// TwinCAT 3 PLC project ProjectMain
// ProgramVersion: 3.1.4023.0
// libraries:
//   Tc2_ControllerToolbox, * (Beckhoff Automation GmbH)
//   Tc2_Math, * (Beckhoff Automation GmbH)
//   Tc2_MC2, * (Beckhoff Automation GmbH)
//   Tc2_MC2_Drive, * (Beckhoff Automation GmbH)
//   Tc2_NCI, * (Beckhoff Automation GmbH)
//   Tc2_NcKinematicTransformation, * (Beckhoff Automation GmbH)
//   Tc2_PlcInterpolation, * (Beckhoff Automation GmbH)
//   Tc2_Standard, * (Beckhoff Automation GmbH)
//   Tc2_System, * (Beckhoff Automation GmbH)
//   Tc2_Utilities, * (Beckhoff Automation GmbH)
//   Tc3_McCollisionAvoidance, * (Beckhoff Automation GmbH)
//   Tc3_McCoordinatedMotion, * (Beckhoff Automation GmbH)
//   Tc3_Module, * (Beckhoff Automation GmbH)
//   Tc3_Vision, * (Beckhoff Automation GmbH)
//   Tc3_XTS_Utility, * (Beckhoff Automation GmbH)
// project tree:
//   DUTs/ DeltaCommands_typ.TcDUT, DeltaMotionParameters_typ.TcDUT, DeltaState_enum.TcDUT, ElevatorState_enum.TcDUT, MachineOperationMode.TcDUT, MainCommands_typ.TcDUT, MainStateAxis_enum.TcDUT, MainState_enum.TcDUT, MotionParameters_typ.TcDUT, MoverCommandType_enum.TcDUT, MoverState_enum.TcDUT, MoveState_t.TcDUT, PickPars_typ.TcDUT, Pucks.TcDUT, SystemCommands_typ.TcDUT, Vector3Position_typ.TcDUT, Visu_typ.TcDUT, Coords.TcDUT, XYParams_typ.TcDUT
//   GVLs/ GVL.TcGVL, GVL_Conveyer.TcGVL, GVL_Vision.TcGVL, GVL_XTS.TcGVL, GVL_XY.TcGVL
//   ITFs/ iDelta.TcIO, iRoute.TcIO
//   / Main1_1.TcTTO, Main2_1.TcTTO, Main3_1.TcTTO, Main4_1.TcTTO, Main5_1.TcTTO
//   Station1%28Codian%29/ Faults1.TcPOU (not stored), fbLoadMoves.TcPOU (not stored), Forces1.TcPOU (not stored), Main1.TcPOU (not stored), Reset1.TcPOU (not stored), Sequence1.TcPOU (not stored)
//   Station1%28Codian%29/Functions/ Delta.TcPOU (not stored), FB_PuckPicked.TcPOU (not stored), Route.TcPOU (not stored)
//   Station2%28XYmover%29/ Faults2.TcPOU (not stored), Forces2.TcPOU (not stored), Main2.TcPOU (not stored), Reset2.TcPOU (not stored), Sequence2.TcPOU (not stored)
//   Station2%28XYmover%29/XY_FBs/ FB_AddAllAxes.TcPOU (not stored), FB_ConveyerTimer.TcPOU (not stored), FB_PowerAll.TcPOU (not stored), FB_ResetAllAxis.TcPOU (not stored), FB_StopAll.TcPOU (not stored)
//   Station3%28Conveyor%29/ Faults3.TcPOU (not stored), Forces3.TcPOU (not stored), Main3.TcPOU (not stored), Reset3.TcPOU (not stored), Sequence3.TcPOU (not stored)
//   Station3%28Conveyor%29/Functions/ FB_ClearConveyer.TcPOU (not stored), FB_ConveyerStop.TcPOU (not stored), FB_PowerConveyer.TcPOU (not stored)
//   Station4%28xts1%29/ Faults4.TcPOU (not stored), Forces4.TcPOU (not stored), Main4.TcPOU (not stored), Reset4.TcPOU (not stored), Sequence4.TcPOU (not stored)
//   Station5%28xts2%29/ Faults5.TcPOU (not stored), Forces5.TcPOU (not stored), Main5.TcPOU (not stored), Reset5.TcPOU (not stored), Sequence5.TcPOU (not stored)
//   Station6%28Vision%29/ Faults6.TcPOU (not stored), Forces6.TcPOU (not stored), Main6.TcPOU (not stored), Reset6.TcPOU (not stored), Sequence6.TcPOU (not stored)
// real-time tasks:
//   TASK PlcTask: cycle T#10ms, priority 20, ADS port 350
//   TASK VnTask ADS (Camera1): cycle T#10ms, priority 16, ADS port 354
//   TASK VnTask ImgAcq (Camera1): cycle T#1ms, priority 10, ADS port 353
//   TASK Job Task: cycle default, priority 32
//   TASK Main1: cycle T#1ms, priority 2, ADS port 351
//   TASK Main2: cycle T#10ms, priority 3, ADS port 355
//   TASK Main3: cycle T#10ms, priority 5, ADS port 356
//   TASK Main4: cycle T#10ms, priority 6, ADS port 357
//   TASK Main5: cycle T#10ms, priority 7, ADS port 358
// motion (NC):
//   TASK NC-Task 1 SAF: cycle T#500us, priority 4, ADS port 501
//   TASK NC-Task 1 SVB: cycle T#10ms, priority 8, ADS port 511
//   AXIS Delta ACS A (id 10)
//     General: UnitName=°
//     Dynamic: Acceleration=2367.9, Deceleration=2367.9, Jerk=7103.7
//     Velo: RefSearch=15.78603, RefSync=15.78603, SlowManual=78.93015, FastManual=473.5809, Fast=1578.603, Maximum=1578.6
//     OtherSettings: AllowMotionCmdToSlave=true
//     encoder EncType=19
//       EncPara: ScaleFactorNumerator=360, ScaleFactorDenominator=23068672, Offset=-24.7313, Inverse=true, MaxCount=#xffffffff
//     drive DrvType=16
//       DrvPara: Inverse=true, MaxCount=#xffffffff, DriveControlDWord=#x00020100
//         Analog: VeloReferenz=1736.4633, TorqueSetpointScale=10, ScaleFactorActTorque=0.1
//         TimeComp: TaskDelayCycles=1
//     controller CtrType=1
//       CtrPara: PriorControlFactor=1
//         Observer: BandWidth=20
//   AXIS Delta ACS B (id 11)
//     General: UnitName=°
//     Dynamic: Acceleration=2367.9, Deceleration=2367.9, Jerk=7103.71
//     Velo: RefSearch=15.78603, RefSync=15.78603, SlowManual=78.93015, FastManual=473.5809, Fast=1578.603, Maximum=1578.6
//     OtherSettings: AllowMotionCmdToSlave=true
//     encoder EncType=19
//       EncPara: ScaleFactorNumerator=360, ScaleFactorDenominator=23068672, Offset=1838.2737, Inverse=true, MaxCount=#xffffffff
//     drive DrvType=16
//       DrvPara: Inverse=true, MaxCount=#xffffffff, DriveControlDWord=#x00020100
//         Analog: VeloReferenz=1736.4633, TorqueSetpointScale=10, ScaleFactorActTorque=0.1
//         TimeComp: TaskDelayCycles=1
//     controller CtrType=1
//       CtrPara: PriorControlFactor=1
//         Observer: BandWidth=20
//   AXIS Delta ACS C (id 12)
//     General: UnitName=°
//     Dynamic: Acceleration=2367.9045, Deceleration=2367.9045, Jerk=7103.7135
//     Velo: RefSearch=15.78603, RefSync=15.78603, SlowManual=78.93015, FastManual=473.5809, Fast=1578.603, Maximum=1578.603
//     OtherSettings: AllowMotionCmdToSlave=true
//     encoder EncType=19
//       EncPara: ScaleFactorNumerator=360, ScaleFactorDenominator=23068672, Offset=9.7019, Inverse=true, MaxCount=#xffffffff
//     drive DrvType=16
//       DrvPara: Inverse=true, MaxCount=#xffffffff, DriveControlDWord=#x00020100
//         Analog: VeloReferenz=1736.4633, TorqueSetpointScale=10, ScaleFactorActTorque=0.1
//         TimeComp: TaskDelayCycles=1
//     controller CtrType=1
//       CtrPara: PriorControlFactor=1
//         Observer: BandWidth=20
//   AXIS Delta MCS X (id 5)
//     Dynamic: Acceleration=12900, Deceleration=12900, Jerk=286914
//     OtherSettings: AllowMotionCmdToSlave=true
//     encoder EncType=1
//       SoftEndMinControl: Enable=true, Range=-100
//       SoftEndMaxControl: Enable=true, Range=100
//     drive DrvType=5
//       Analog: VeloReferenz=500, TorqueSetpointScale=10, ScaleFactorActTorque=0.1
//       TimeComp: TaskDelayCycles=1
//     controller CtrType=1
//       CtrPara: PriorControlFactor=1
//         Observer: BandWidth=20
//   AXIS Delta MCS Y (id 6)
//     Dynamic: Acceleration=13125, Deceleration=13125, Jerk=275625
//     OtherSettings: AllowMotionCmdToSlave=true
//     encoder EncType=1
//       SoftEndMinControl: Enable=true, Range=-80
//       SoftEndMaxControl: Enable=true, Range=150
//     drive DrvType=5
//       Analog: VeloReferenz=500, TorqueSetpointScale=10, ScaleFactorActTorque=0.1
//       TimeComp: TaskDelayCycles=1
//     controller CtrType=1
//       CtrPara: PriorControlFactor=1
//         Observer: BandWidth=20
//   AXIS Delta MCS Z (id 7)
//     Dynamic: Acceleration=15100, Deceleration=15100, Jerk=223539
//     OtherSettings: AllowMotionCmdToSlave=true
//     encoder EncType=1
//       EncPara: Offset=-250
//         SoftEndMinControl: Range=-60
//         SoftEndMaxControl: Enable=true, Range=25
//     drive DrvType=5
//       Analog: VeloReferenz=500, TorqueSetpointScale=10, ScaleFactorActTorque=0.1
//       TimeComp: TaskDelayCycles=1
//     controller CtrType=1
//       CtrPara: PriorControlFactor=1
//         Observer: BandWidth=20
//   AXIS Y (id 1)
//     Dynamic: Acceleration=540.1395, Deceleration=540.1395, Jerk=1620.4185
//     Velo: RefSearch=3.60093, RefSync=3.60093, SlowManual=18.00465, FastManual=108.0279, Fast=360.093, Maximum=360.093
//     OtherSettings: AllowMotionCmdToSlave=true
//     encoder EncType=19
//       EncPara: ScaleFactorNumerator=4, ScaleFactorDenominator=1048576, Offset=7764.81834411621, MaxCount=#xffffffff, ReferenceSystem=1
//         SoftEndMinControl: Enable=true
//         SoftEndMaxControl: Enable=true, Range=385
//     drive DrvType=16
//       DrvPara: MaxCount=#xffffffff, DriveControlDWord=#x00020100
//         Analog: VeloReferenz=396.1023, VeloScale=32, TorqueSetpointScale=10, ScaleFactorActTorque=0.1
//         TimeComp: TaskDelayCycles=1
//     controller CtrType=1
//       CtrPara: PriorControlFactor=1
//         Observer: BandWidth=20
//   AXIS X (id 2)
//     Dynamic: Acceleration=540.9, Deceleration=540.9, Jerk=1622.7
//     Velo: RefSearch=3.606, RefSync=3.606, SlowManual=18.03, FastManual=108.18, Fast=360.6, Maximum=360.6
//     OtherSettings: AllowMotionCmdToSlave=true
//     encoder EncType=19
//       EncPara: ScaleFactorNumerator=4, ScaleFactorDenominator=1048576, MaxCount=#xffffffff, ReferenceSystem=3
//         SoftEndMinControl: Enable=true
//         SoftEndMaxControl: Enable=true, Range=200
//     drive DrvType=16
//       DrvPara: MaxCount=#xffffffff, DriveControlDWord=#x00020100
//         Analog: VeloReferenz=396.66, VeloScale=32, TorqueSetpointScale=10, ScaleFactorActTorque=0.1
//         TimeComp: TaskDelayCycles=1
//     controller CtrType=1
//       CtrPara: PriorControlFactor=1
//         Observer: BandWidth=20
//   AXIS X Slave (id 3)
//     Dynamic: Acceleration=524.2, Deceleration=524.2, Jerk=1572.6
//     Velo: RefSearch=3.49466666666667, RefSync=3.49466666666667, SlowManual=17.4733333333333, FastManual=104.84, Fast=349.466666666667, Maximum=349.466666666667
//     OtherSettings: AllowMotionCmdToSlave=true
//     encoder EncType=19
//       EncPara: ScaleFactorNumerator=4, ScaleFactorDenominator=1048576, Offset=-2512.61434173584, MaxCount=#xffffffff, ReferenceSystem=3
//         SoftEndMinControl: Enable=true
//         SoftEndMaxControl: Enable=true, Range=200
//     drive DrvType=16
//       DrvPara: MaxCount=#xffffffff, DriveControlDWord=#x00020100
//         Analog: VeloReferenz=384.413333333333, VeloScale=32, TorqueSetpointScale=10, ScaleFactorActTorque=0.1
//         TimeComp: TaskDelayCycles=1
//     controller CtrType=1
//       CtrPara: PriorControlFactor=1
//         Observer: BandWidth=20
//   AXIS ConveyorAxis (id 4)
//     General: UnitName=°
//     Dynamic: AccelerationMaximum=48963.411, DecelerationMaximum=48963.411, Acceleration=48681, Deceleration=48681, Jerk=146043
//     Velo: RefSearch=324.54, RefSync=324.54, SlowManual=1622.7, FastManual=9736.2, Fast=32454, Maximum=32454
//     OtherSettings: AllowMotionCmdToSlave=true
//     encoder EncType=19
//       EncPara: ScaleFactorNumerator=360, ScaleFactorDenominator=1048576, MaxCount=#xffffffff
//     drive DrvType=16
//       DrvPara: MaxCount=#xffffffff, DriveControlDWord=#x00020100
//         Analog: VeloReferenz=35699.4, VeloScale=32, TorqueSetpointScale=10, ScaleFactorActTorque=0.1
//         TimeComp: TaskDelayCycles=1
//     controller CtrType=1
//       CtrPara: PriorControlFactor=1
//         PosDiffControl: Enable=false, Range=25
//         Observer: BandWidth=20
// I/O:
//   DEVICE Device 3 (EtherCAT), AmsNetId 169.254.124.141.4.1
//     Term 1 (EK1100) [EK1100 EtherCAT Coupler (2A E-Bus)]
//       Term 2 (EL1918) [EL1918, 8Ch. Safety Input 24V, TwinSAFE]
//         modules: Module 2 (FSLOGIC)
//       Term 3 (EL1008) [EL1008 8Ch. Dig. Input 24V, 3ms]
//       Term 4 (EL2904) [EL2904, 4 Ch. Safety Output 24V, 0.5A, TwinSAFE]
//         modules: Module 1 (FSOES), Module 2 (DO)
//       Term 5 (EL2008) [EL2008 8Ch. Dig. Output 24V, 0.5A]
//       Term 6 (EL7201-9014) [EL7201-9014 1Ch. MDP742 Servo motor output stage with OCT (50V, 4A)  and STO input]
//         startup 32785:27 := 23150000 // DRV Motor Settings / Motor speed limitation
//         startup 32784:19 := B200 // DRV Amplifier Settings / Current loop proportional gain
//         startup 32784:18 := 0500 // DRV Amplifier Settings / Current loop integral time
//         startup 32784:21 := 25000000 // DRV Amplifier Settings / Velocity loop proportional gain
//         startup 32784:20 := 96000000 // DRV Amplifier Settings / Velocity loop integral time
//         startup 32768:1 := 00 // FB Settings / Invert feedback direction
//       Term 7 (EL7211-9014) [EL7211-9014 1Ch. MDP742 Servo motor output stage with OCT (50V, 4.5A RMS) and STO input]
//         startup 32785:21 := 0E01 // DRV Motor Settings / Commutation offset
//         startup 32786:19 := F401 // DRV Brake Settings / Emergency application timeout
//         startup 32784:51 := 0A00 // DRV Amplifier Settings / Stand still window
//         startup 32785:27 := 21150000 // DRV Motor Settings / Motor speed limitation
//         startup 32784:19 := B200 // DRV Amplifier Settings / Current loop proportional gain
//         startup 32784:18 := 0500 // DRV Amplifier Settings / Current loop integral time
//         startup 32784:21 := 48000000 // DRV Amplifier Settings / Velocity loop proportional gain
//         startup 32784:20 := 96000000 // DRV Amplifier Settings / Velocity loop integral time
//         startup 32768:1 := 00 // FB Settings / Invert feedback direction
//       Term 22 (EL7211-9014) [EL7211-9014 1Ch. MDP742 Servo motor output stage with OCT (50V, 4.5A RMS) and STO input]
//         startup 32784:18 := 0A00
//         startup 32784:19 := 6400
//         startup 32784:20 := 32000000
//         startup 32784:21 := 96000000
//         startup 32784:51 := 0A00
//         startup 32785:17 := 98210000
//         startup 32785:18 := 960A0000
//         startup 32785:19 := 03
//         startup 32785:21 := 0E01
//         startup 32785:22 := 46000000
//         startup 32785:24 := 39000000
//         startup 32785:25 := 0F00
//         startup 32785:27 := FF120000
//         startup 32785:45 := 5501
//         startup 32786:17 := 0800
//         startup 32786:18 := 0E00
//         startup 32786:19 := F401
//       Term 9 (EL7211-9014) [EL7211-9014 1Ch. MDP742 Servo motor output stage with OCT (50V, 4.5A RMS) and STO input]
//         startup 32785:21 := 0E01 // DRV Motor Settings / Commutation offset
//         startup 32786:19 := F401 // DRV Brake Settings / Emergency application timeout
//         startup 32784:51 := 0A00 // DRV Amplifier Settings / Stand still window
//         startup 32785:27 := 21150000 // DRV Motor Settings / Motor speed limitation
//         startup 32784:19 := B200 // DRV Amplifier Settings / Current loop proportional gain
//         startup 32784:18 := 0500 // DRV Amplifier Settings / Current loop integral time
//         startup 32784:21 := 48000000 // DRV Amplifier Settings / Velocity loop proportional gain
//         startup 32784:20 := 96000000 // DRV Amplifier Settings / Velocity loop integral time
//         startup 32768:1 := 00 // FB Settings / Invert feedback direction
//       Term 13 (EL9011) [EL9011 End Terminal]
//     Term 10 (AX8620-0000-0103) [AX8620-0000-0103]
//       Drive 11 (AX8108-0100-0104) [AX8108-0100-0104 (1Ch. 8A servo axis, STO)]
//         modules: Device, Device, Device, Device, Device, Device, Device, Device, Device, Device, Device (Safety), Device, Device, Device, Device, Device, Device, Device, Device, Device, Device, Device, Device, Device, Device, Device, Device, Device, Device, Device, Device, Ch A, Ch A, Ch A, Ch A, Ch A, Ch A, Ch A, Ch A, Ch A, Ch A, Ch A, Ch A, Ch A, Ch A, Ch A, Ch A, Ch A, Ch A, Ch A, Ch A, Ch A, Ch A, Ch A, Ch A, Ch A, Ch A, Ch A
//         startup 12992:1 := 414D383033312D78467830 // Ch A Motor parameters / Configured motor type
//         startup 24768:0 := FEFF // Ch A Interpolation sub mode select
//         startup 13000:5 := 0200 // Ch A Motor thermal model / Reaction
//         startup 13000:6 := 0000C841 // Ch A Motor thermal model / Partial fraction factor
//         startup 12992:12 := 00A00C46 // Ch A Motor parameters / Motor rated speed
//         startup 12992:13 := 2731A83F // Ch A Motor parameters / Motor rated torque
//         startup 24694:0 := 7A050000 // Ch A Motor standstill torque
//         startup 24800:0 := D007 // Ch A Positive torque/force limit value
//         startup 24801:0 := D007 // Ch A Negative torque/force limit value
//         startup 12288:6 := 4158383130382D303130302D30303030 // Ch A AxisMain parameters / Configured drive type
//         startup 12867:1 := CDCC4C40 // Ch A TorqueCtrl parameters / Configured channel rated current
//         startup 12867:2 := 9A991941 // Ch A TorqueCtrl parameters / Configured channel peak current
//         startup 24672:0 := 08 // Ch A Modes of operation
//         startup 12864:1 := 60CE3E42 // Ch A TorqueCtrl parameters mappable / Torque control proportional gain q
//         startup 12864:2 := 8A0E7C39 // Ch A TorqueCtrl parameters mappable / Torque control integral action time q
//         startup 12608:1 := 9C67B13C // Ch A VeloCtrl parameters mappable / Velocity control proportional gain
//         startup 12608:2 := 6F12033C // Ch A VeloCtrl parameters mappable / Velocity control integral action time
//         startup 12608:3 := 00980546 // Ch A VeloCtrl parameters mappable / Bipolar velocity limit value
//         startup 12992:15 := 0100 // Ch A Motor parameters / Motor temperature sensor connection
//         startup 12611:4 := 0400 // Ch A VeloCtrl observer / Observer type
//         startup 24672:0 := 08 // Ch A Modes of operation
//         startup 12296:2 := 00 // Ch A AxisMain parameters encoder polarity / Primary encoder actual values
//       Drive 12 (AX8206-0210-0104) [AX8206-0210-0104 (2Ch. 6A servo axis, safe-motion, multi-FB)]
//         modules: Device, Device, Device, Device, Device, Device, Device, Device, Device, Device, Device (Safety), Device, Device, Device, Device, Device, Device, Device, Device, Device, Device, Device, Device, Device, Device, Device, Device, Device, Device, Device, Device, Ch A, Ch A, Ch A, Ch A, Ch A, Ch A, Ch A, Ch A, Ch A, Ch A, Ch A, Ch A, Ch A, Ch A, Ch A, Ch A, Ch A, Ch A, Ch A, Ch A, Ch A, Ch A, Ch A, Ch A, Ch A, Ch A, Ch B, Ch B, Ch B, Ch B, Ch B, Ch B, Ch B, Ch B, Ch B, Ch B, Ch B, Ch B, Ch B, Ch B, Ch B, Ch B, Ch B, Ch B, Ch B, Ch B, Ch B, Ch B, Ch B, Ch B, Ch B, Ch B
//         startup 12992:1 := 414D383033312D78467830 // Ch A Motor parameters / Configured motor type
//         startup 24768:0 := FEFF // Ch A Interpolation sub mode select
//         startup 13000:5 := 0200 // Ch A Motor thermal model / Reaction
//         startup 13000:6 := 0000C841 // Ch A Motor thermal model / Partial fraction factor
//         startup 12992:12 := 00A00C46 // Ch A Motor parameters / Motor rated speed
//         startup 12992:13 := 2731A83F // Ch A Motor parameters / Motor rated torque
//         startup 24694:0 := 7A050000 // Ch A Motor standstill torque
//         startup 24800:0 := D007 // Ch A Positive torque/force limit value
//         startup 24801:0 := D007 // Ch A Negative torque/force limit value
//         startup 12288:6 := 4158383230362D303231302D30303030 // Ch A AxisMain parameters / Configured drive type
//         startup 12867:1 := CDCC4C40 // Ch A TorqueCtrl parameters / Configured channel rated current
//         startup 12867:2 := 9A991941 // Ch A TorqueCtrl parameters / Configured channel peak current
//         startup 24672:0 := 08 // Ch A Modes of operation
//         startup 12864:1 := 60CE3E42 // Ch A TorqueCtrl parameters mappable / Torque control proportional gain q
//         startup 12864:2 := 8A0E7C39 // Ch A TorqueCtrl parameters mappable / Torque control integral action time q
//         startup 12608:1 := 9C67B13C // Ch A VeloCtrl parameters mappable / Velocity control proportional gain
//         startup 12608:2 := 6F12033C // Ch A VeloCtrl parameters mappable / Velocity control integral action time
//         startup 12608:3 := 00980546 // Ch A VeloCtrl parameters mappable / Bipolar velocity limit value
//         startup 12992:15 := 0100 // Ch A Motor parameters / Motor temperature sensor connection
//         startup 12611:4 := 0400 // Ch A VeloCtrl observer / Observer type
//         startup 24672:0 := 08 // Ch A Modes of operation
//         startup 12296:2 := 00 // Ch A AxisMain parameters encoder polarity / Primary encoder actual values
//         startup 14016:1 := 414D383033312D78467830 // Ch B Motor parameters / Configured motor type
//         startup 26816:0 := FEFF // Ch B Interpolation sub mode select
//         startup 14024:5 := 0200 // Ch B Motor thermal model / Reaction
//         startup 14024:6 := 0000C841 // Ch B Motor thermal model / Partial fraction factor
//         startup 14016:12 := 00A00C46 // Ch B Motor parameters / Motor rated speed
//         startup 14016:13 := 2731A83F // Ch B Motor parameters / Motor rated torque
//         startup 26742:0 := 7A050000 // Ch B Motor standstill torque
//         startup 26848:0 := D007 // Ch B Positive torque/force limit value
//         startup 26849:0 := D007 // Ch B Negative torque/force limit value
//         startup 13312:6 := 4158383230362D303231302D30303030 // Ch B AxisMain parameters / Configured drive type
//         startup 13891:1 := CDCC4C40 // Ch B TorqueCtrl parameters / Configured channel rated current
//         startup 13891:2 := 9A991941 // Ch B TorqueCtrl parameters / Configured channel peak current
//         startup 26720:0 := 08 // Ch B Modes of operation
//         startup 13888:1 := 60CE3E42 // Ch B TorqueCtrl parameters mappable / Torque control proportional gain q
//         startup 13888:2 := 8A0E7C39 // Ch B TorqueCtrl parameters mappable / Torque control integral action time q
//         startup 13632:1 := 9C67B13C // Ch B VeloCtrl parameters mappable / Velocity control proportional gain
//         startup 13632:2 := 6F12033C // Ch B VeloCtrl parameters mappable / Velocity control integral action time
//         startup 13632:3 := 00980546 // Ch B VeloCtrl parameters mappable / Bipolar velocity limit value
//         startup 14016:15 := 0100 // Ch B Motor parameters / Motor temperature sensor connection
//         startup 13635:4 := 0400 // Ch B VeloCtrl observer / Observer type
//         startup 26720:0 := 08 // Ch B Modes of operation
//         startup 13320:2 := 00 // Ch B AxisMain parameters encoder polarity / Primary encoder actual values
//       Term 14 (EL9011) [EL9011 End Terminal]
//   DEVICE Device 1 (EtherCAT Automation Protocol), AmsNetId 169.254.124.141.2.1
//     Box 8 (Publisher)
//     Box 15 (Subscriber)
// variable links:
//   Device 3 (EtherCAT) <-> Device 3 (EtherCAT)/Term 1 (EK1100)/Term 2 (EL1918)
//     Term 1 (EK1100)/Term 4 (EL2904)/Module 1 (FSOES)/RxPDO/FSOE <-> ConnectionInputs/Message_4 TxPDO
//     Term 10 (AX8620-0000-0103)/Drive 12 (AX8206-0210-0104)/Device (Safety)/FSoE Slave Connection 1 Slave Message/FSOE <-> ConnectionOutputs/Message_6 RxPDO
//   Device 3 (EtherCAT) <-> Device 3 (EtherCAT)/Term 1 (EK1100)/Term 4 (EL2904)
//     Term 1 (EK1100)/Term 2 (EL1918)/ConnectionOutputs/Message_4 RxPDO <-> Module 1 (FSOES)/TxPDO/FSOE
//   Device 3 (EtherCAT) <-> Device 3 (EtherCAT)/Term 10 (AX8620-0000-0103)
//     Term 10 (AX8620-0000-0103)/Drive 11 (AX8108-0100-0104)/Device/DeviceMain Outputs/Power supply controlword <-> PSM Controlword for axis/Controlword for axis
//     Term 10 (AX8620-0000-0103)/Drive 12 (AX8206-0210-0104)/Device/DeviceMain Outputs/Power supply controlword <-> PSM Controlword for axis/Controlword for axis
//   Device 3 (EtherCAT) <-> Device 3 (EtherCAT)/Term 10 (AX8620-0000-0103)/Drive 11 (AX8108-0100-0104)
//     Term 1 (EK1100)/Term 2 (EL1918)/ConnectionInputs/Message_5 TxPDO <-> Device (Safety)/FSoE Slave Connection 1 Master Message/FSOE
//     Term 1 (EK1100)/Term 2 (EL1918)/ConnectionOutputs/Message_5 RxPDO <-> Device (Safety)/FSoE Slave Connection 1 Slave Message/FSOE
//   Device 3 (EtherCAT) <-> Device 3 (EtherCAT)/Term 10 (AX8620-0000-0103)/Drive 12 (AX8206-0210-0104)
//     Term 1 (EK1100)/Term 2 (EL1918)/ConnectionInputs/Message_6 TxPDO <-> Device (Safety)/FSoE Slave Connection 1 Master Message/FSOE
//   NC-Task 1 SAF/Axes/ConveyorAxis <-> Device 3 (EtherCAT)/Term 1 (EK1100)/Term 9 (EL7211-9014)
//     Drive/Inputs/In/nDataIn1 <-> DRV Following error actual value/Following error actual value
//     Drive/Inputs/In/nDcOutputTime <-> InfoData/DcOutputShift
//     Drive/Inputs/In/nState1 <-> DRV Statusword/Statusword
//     Drive/Inputs/In/nState2 <-> DRV Statusword/Statusword @bit 8
//     Drive/Inputs/In/nState4 @bit 1 <-> WcState/InputToggle
//     Drive/Inputs/In/nState4 <-> WcState/WcState
//     Drive/Outputs/Out/nCtrl1 <-> DRV Controlword/Controlword
//     Drive/Outputs/Out/nCtrl2 <-> DRV Controlword/Controlword @bit 8
//     Drive/Outputs/Out/nDataOut1 <-> DRV Target position/Target position
//     Drive/Outputs/Out/nDataOut2 <-> DRV Target velocity/Target velocity
//     Enc/Inputs/In/nDataIn1 <-> FB Position/Position
//     Enc/Inputs/In/nDcInputTime <-> InfoData/DcInputShift
//     Enc/Inputs/In/nState4 @bit 1 <-> WcState/InputToggle
//     Enc/Inputs/In/nState4 <-> WcState/WcState
//   NC-Task 1 SAF/Axes/Delta ACS A <-> Device 3 (EtherCAT)/Term 10 (AX8620-0000-0103)/Drive 11 (AX8108-0100-0104)
//     Drive/Inputs/In/nDataIn1 <-> Ch A/Ch A PositionControl Inputs/Ch A Following error actual value
//     Drive/Inputs/In/nDcOutputTime <-> InfoData/DcOutputShift
//     Drive/Inputs/In/nState1 <-> Ch A/Ch A AxisMain Inputs/Ch A Statusword
//     Drive/Inputs/In/nState2 <-> Ch A/Ch A AxisMain Inputs/Ch A Statusword @bit 8
//     Drive/Inputs/In/nState4 @bit 1 <-> WcState/InputToggle0
//     Drive/Inputs/In/nState4 <-> WcState/WcState0
//     Drive/Outputs/Out/nCtrl1 <-> Ch A/Ch A AxisMain Outputs/Ch A Controlword
//     Drive/Outputs/Out/nCtrl2 <-> Ch A/Ch A AxisMain Outputs/Ch A Controlword @bit 8
//     Drive/Outputs/Out/nDataOut1 <-> Ch A/Ch A Interpolator Outputs/Ch A Target position
//     Drive/Outputs/Out/nDataOut2 <-> Ch A/Ch A Interpolator Outputs/Ch A Target velocity
//     Enc/Inputs/In/nDataIn1 <-> Ch A/Ch A AxisMain Inputs/Ch A Position actual value
//     Enc/Inputs/In/nDcInputTime <-> InfoData/DcInputShift
//     Enc/Inputs/In/nState2 @bit 5 <-> Ch A/Ch A AxisMain Inputs/Position actual value invalid
//     Enc/Inputs/In/nState4 @bit 1 <-> WcState/InputToggle0
//     Enc/Inputs/In/nState4 <-> WcState/WcState0
//   NC-Task 1 SAF/Axes/Delta ACS B <-> Device 3 (EtherCAT)/Term 10 (AX8620-0000-0103)/Drive 12 (AX8206-0210-0104)
//     Drive/Inputs/In/nDataIn1 <-> Ch A/Ch A PositionControl Inputs/Ch A Following error actual value
//     Drive/Inputs/In/nDcOutputTime <-> InfoData/DcOutputShift
//     Drive/Inputs/In/nState1 <-> Ch A/Ch A AxisMain Inputs/Ch A Statusword
//     Drive/Inputs/In/nState2 <-> Ch A/Ch A AxisMain Inputs/Ch A Statusword @bit 8
//     Drive/Inputs/In/nState4 @bit 1 <-> WcState/InputToggle0
//     Drive/Inputs/In/nState4 <-> WcState/WcState0
//     Drive/Outputs/Out/nCtrl1 <-> Ch A/Ch A AxisMain Outputs/Ch A Controlword
//     Drive/Outputs/Out/nCtrl2 <-> Ch A/Ch A AxisMain Outputs/Ch A Controlword @bit 8
//     Drive/Outputs/Out/nDataOut1 <-> Ch A/Ch A Interpolator Outputs/Ch A Target position
//     Drive/Outputs/Out/nDataOut2 <-> Ch A/Ch A Interpolator Outputs/Ch A Target velocity
//     Enc/Inputs/In/nDataIn1 <-> Ch A/Ch A AxisMain Inputs/Ch A Position actual value
//     Enc/Inputs/In/nDcInputTime <-> InfoData/DcInputShift
//     Enc/Inputs/In/nState2 @bit 5 <-> Ch A/Ch A AxisMain Inputs/Position actual value invalid
//     Enc/Inputs/In/nState4 @bit 1 <-> WcState/InputToggle0
//     Enc/Inputs/In/nState4 <-> WcState/WcState0
//   NC-Task 1 SAF/Axes/Delta ACS C <-> Device 3 (EtherCAT)/Term 10 (AX8620-0000-0103)/Drive 12 (AX8206-0210-0104)
//     Drive/Inputs/In/nDataIn1 <-> Ch B/Ch B PositionControl Inputs/Ch B Following error actual value
//     Drive/Inputs/In/nDcOutputTime <-> InfoData/DcOutputShift
//     Drive/Inputs/In/nState1 <-> Ch B/Ch B AxisMain Inputs/Ch B Statusword
//     Drive/Inputs/In/nState2 <-> Ch B/Ch B AxisMain Inputs/Ch B Statusword @bit 8
//     Drive/Inputs/In/nState4 @bit 1 <-> WcState/InputToggle0
//     Drive/Inputs/In/nState4 <-> WcState/WcState0
//     Drive/Outputs/Out/nCtrl1 <-> Ch B/Ch B AxisMain Outputs/Ch B Controlword
//     Drive/Outputs/Out/nCtrl2 <-> Ch B/Ch B AxisMain Outputs/Ch B Controlword @bit 8
//     Drive/Outputs/Out/nDataOut1 <-> Ch B/Ch B Interpolator Outputs/Ch B Target position
//     Drive/Outputs/Out/nDataOut2 <-> Ch B/Ch B Interpolator Outputs/Ch B Target velocity
//     Enc/Inputs/In/nDataIn1 <-> Ch B/Ch B AxisMain Inputs/Ch B Position actual value
//     Enc/Inputs/In/nDcInputTime <-> InfoData/DcInputShift
//     Enc/Inputs/In/nState2 @bit 5 <-> Ch B/Ch B AxisMain Inputs/Position actual value invalid
//     Enc/Inputs/In/nState4 @bit 1 <-> WcState/InputToggle0
//     Enc/Inputs/In/nState4 <-> WcState/WcState0
//   NC-Task 1 SAF/Axes/X <-> Device 3 (EtherCAT)/Term 1 (EK1100)/Term 7 (EL7211-9014)
//     Drive/Inputs/In/nDataIn1 <-> DRV Following error actual value/Following error actual value
//     Drive/Inputs/In/nDcOutputTime <-> InfoData/DcOutputShift
//     Drive/Inputs/In/nState1 <-> DRV Statusword/Statusword
//     Drive/Inputs/In/nState2 <-> DRV Statusword/Statusword @bit 8
//     Drive/Inputs/In/nState4 @bit 1 <-> WcState/InputToggle
//     Drive/Inputs/In/nState4 <-> WcState/WcState
//     Drive/Outputs/Out/nCtrl1 <-> DRV Controlword/Controlword
//     Drive/Outputs/Out/nCtrl2 <-> DRV Controlword/Controlword @bit 8
//     Drive/Outputs/Out/nDataOut1 <-> DRV Target position/Target position
//     Drive/Outputs/Out/nDataOut2 <-> DRV Target velocity/Target velocity
//     Enc/Inputs/In/nDataIn1 <-> FB Position/Position
//     Enc/Inputs/In/nDcInputTime <-> InfoData/DcInputShift
//     Enc/Inputs/In/nState4 @bit 1 <-> WcState/InputToggle
//     Enc/Inputs/In/nState4 <-> WcState/WcState
//   NC-Task 1 SAF/Axes/X Slave <-> Device 3 (EtherCAT)/Term 1 (EK1100)/Term 22 (EL7211-9014)
//     Drive/Inputs/In/nDataIn1 <-> DRV Following error actual value/Following error actual value
//     Drive/Inputs/In/nDcOutputTime <-> InfoData/DcOutputShift
//     Drive/Inputs/In/nState1 <-> DRV Statusword/Statusword
//     Drive/Inputs/In/nState2 <-> DRV Statusword/Statusword @bit 8
//     Drive/Inputs/In/nState4 @bit 1 <-> WcState/InputToggle
//     Drive/Inputs/In/nState4 <-> WcState/WcState
//     Drive/Outputs/Out/nCtrl1 <-> DRV Controlword/Controlword
//     Drive/Outputs/Out/nCtrl2 <-> DRV Controlword/Controlword @bit 8
//     Drive/Outputs/Out/nDataOut1 <-> DRV Target position/Target position
//     Drive/Outputs/Out/nDataOut2 <-> DRV Target velocity/Target velocity
//     Enc/Inputs/In/nDataIn1 <-> FB Position/Position
//     Enc/Inputs/In/nDcInputTime <-> InfoData/DcInputShift
//     Enc/Inputs/In/nState4 @bit 1 <-> WcState/InputToggle
//     Enc/Inputs/In/nState4 <-> WcState/WcState
//   NC-Task 1 SAF/Axes/Y <-> Device 3 (EtherCAT)/Term 1 (EK1100)/Term 6 (EL7201-9014)
//     Drive/Inputs/In/nDataIn1 <-> DRV Following error actual value/Following error actual value
//     Drive/Inputs/In/nDcOutputTime <-> InfoData/DcOutputShift
//     Drive/Inputs/In/nState1 <-> DRV Statusword/Statusword
//     Drive/Inputs/In/nState2 <-> DRV Statusword/Statusword @bit 8
//     Drive/Inputs/In/nState4 @bit 1 <-> WcState/InputToggle
//     Drive/Inputs/In/nState4 <-> WcState/WcState
//     Drive/Outputs/Out/nCtrl1 <-> DRV Controlword/Controlword
//     Drive/Outputs/Out/nCtrl2 <-> DRV Controlword/Controlword @bit 8
//     Drive/Outputs/Out/nDataOut1 <-> DRV Target position/Target position
//     Drive/Outputs/Out/nDataOut2 <-> DRV Target velocity/Target velocity
//     Enc/Inputs/In/nDataIn1 <-> FB Position/Position
//     Enc/Inputs/In/nDcInputTime <-> InfoData/DcInputShift
//     Enc/Inputs/In/nState4 @bit 1 <-> WcState/InputToggle
//     Enc/Inputs/In/nState4 <-> WcState/WcState
//   ProjectMain/ProjectMain Instance <-> Device 1 (EtherCAT Automation Protocol)/Box 15 (Subscriber)
//     Main1_1 Inputs/GVL_XTS.mover0InPosition <-> mover0InPosition/Inputs/VarData
//     Main2_1 Inputs/GVL_XTS.moversInPosition[1] <-> moversInPosition/Inputs/VarData[1]
//     Main2_1 Inputs/GVL_XTS.moversInPosition[2] <-> moversInPosition/Inputs/VarData[2]
//     Main2_1 Inputs/GVL_XTS.moversInPosition[3] <-> moversInPosition/Inputs/VarData[3]
//     Main5_1 Inputs/GVL_XTS.moversReleased[1] <-> moversReleased/Inputs/VarData[1]
//     Main5_1 Inputs/GVL_XTS.moversReleased[2] <-> moversReleased/Inputs/VarData[2]
//     Main5_1 Inputs/GVL_XTS.moversReleased[3] <-> moversReleased/Inputs/VarData[3]
//   ProjectMain/ProjectMain Instance <-> Device 1 (EtherCAT Automation Protocol)/Box 8 (Publisher)
//     Main1_1 Outputs/GVL_XTS.bDeltaRelease <-> bDeltaRelease/Outputs/VarData
//     Main2_1 Outputs/GVL_XTS.moversRelease <-> moversRelease/Outputs/VarData[1]
//     Main2_1 Outputs/GVL_XTS.moversRelease @bit 8 <-> moversRelease/Outputs/VarData[2]
//     Main2_1 Outputs/GVL_XTS.moversRelease @bit 16 <-> moversRelease/Outputs/VarData[3]
//     Main4_1 Outputs/GVL_XTS.XTS_Disable <-> XTS_Disable/Outputs/VarData
//     Main4_1 Outputs/GVL_XTS.XTS_Enable <-> XTS_Enable/Outputs/VarData
//     Main4_1 Outputs/GVL_XTS.XTS_Start <-> XTS_Start/Outputs/VarData
//     Main4_1 Outputs/GVL_XTS.XTS_Stop <-> XTS_Stop/Outputs/VarData
//   ProjectMain/ProjectMain Instance <-> Device 3 (EtherCAT)/Term 1 (EK1100)/Term 3 (EL1008)
//     Main1_1 Inputs/GVL_Conveyer.bSensor <-> Channel 7/GVL_Conveyer.bSensor
//   ProjectMain/ProjectMain Instance <-> Device 3 (EtherCAT)/Term 1 (EK1100)/Term 5 (EL2008)
//     Main1_1 Outputs/Main1.Sequence1.Delta.AirVariable <-> Channel 8/Main1.Sequence.Delta.AirVariable
//     Main2_1 Outputs/GVL_XY.bAirEnable <-> Channel 2/GantryVacuum
//     Main2_1 Outputs/GVL_XY.bPullUp <-> Channel 4/GrantryPushUp
//     Main2_1 Outputs/GVL_XY.bPushDown <-> Channel 6/GantryPushDown
//   ProjectMain/ProjectMain Instance <-> NC-Task 1 SAF/Axes/ConveyorAxis
//     Main2_1 Inputs/GVL_Conveyer.ConveyerAxis.NcToPlc <-> Outputs/ToPlc
//     Main2_1 Outputs/GVL_Conveyer.ConveyerAxis.PlcToNc <-> Inputs/FromPlc
//   ProjectMain/ProjectMain Instance <-> NC-Task 1 SAF/Axes/Delta ACS A
//     Main1_1 Inputs/Main1.Sequence1.Delta.ACS_A_REF.NcToPlc <-> Outputs/ToPlc
//     Main1_1 Outputs/Main1.Sequence1.Delta.ACS_A_REF.PlcToNc <-> Inputs/FromPlc
//   ProjectMain/ProjectMain Instance <-> NC-Task 1 SAF/Axes/Delta ACS B
//     Main1_1 Inputs/Main1.Sequence1.Delta.ACS_B_REF.NcToPlc <-> Outputs/ToPlc
//     Main1_1 Outputs/Main1.Sequence1.Delta.ACS_B_REF.PlcToNc <-> Inputs/FromPlc
//   ProjectMain/ProjectMain Instance <-> NC-Task 1 SAF/Axes/Delta ACS C
//     Main1_1 Inputs/Main1.Sequence1.Delta.ACS_C_REF.NcToPlc <-> Outputs/ToPlc
//     Main1_1 Outputs/Main1.Sequence1.Delta.ACS_C_REF.PlcToNc <-> Inputs/FromPlc
//   ProjectMain/ProjectMain Instance <-> NC-Task 1 SAF/Axes/Delta MCS X
//     Main1_1 Inputs/Main1.Sequence1.Delta.MCS_X_REF.NcToPlc <-> Outputs/ToPlc
//     Main1_1 Outputs/Main1.Sequence1.Delta.MCS_X_REF.PlcToNc <-> Inputs/FromPlc
//   ProjectMain/ProjectMain Instance <-> NC-Task 1 SAF/Axes/Delta MCS Y
//     Main1_1 Inputs/Main1.Sequence1.Delta.MCS_Y_REF.NcToPlc <-> Outputs/ToPlc
//     Main1_1 Outputs/Main1.Sequence1.Delta.MCS_Y_REF.PlcToNc <-> Inputs/FromPlc
//   ProjectMain/ProjectMain Instance <-> NC-Task 1 SAF/Axes/Delta MCS Z
//     Main1_1 Inputs/Main1.Sequence1.Delta.MCS_Z_REF.NcToPlc <-> Outputs/ToPlc
//     Main1_1 Outputs/Main1.Sequence1.Delta.MCS_Z_REF.PlcToNc <-> Inputs/FromPlc
//   ProjectMain/ProjectMain Instance <-> NC-Task 1 SAF/Axes/X
//     Main2_1 Inputs/GVL_XY.stAxis[1].NcToPlc <-> Outputs/ToPlc
//     Main2_1 Outputs/GVL_XY.stAxis[1].PlcToNc <-> Inputs/FromPlc
//   ProjectMain/ProjectMain Instance <-> NC-Task 1 SAF/Axes/X Slave
//     Main2_1 Inputs/GVL_XY.stSlaveAxis[1].NcToPlc <-> Outputs/ToPlc
//     Main2_1 Outputs/GVL_XY.stSlaveAxis[1].PlcToNc <-> Inputs/FromPlc
//   ProjectMain/ProjectMain Instance <-> NC-Task 1 SAF/Axes/Y
//     Main2_1 Inputs/GVL_XY.stAxis[2].NcToPlc <-> Outputs/ToPlc
//     Main2_1 Outputs/GVL_XY.stAxis[2].PlcToNc <-> Inputs/FromPlc
//   ProjectMain/ProjectMain Instance <-> NC-Task 1 SAF/Channel_Kinnematics
//     Main1_1 Inputs/Main1.Sequence1.Delta.internalKinChanNCtoPLC <-> Outputs/Main1.Sequence.Delta.internalKinChanNCtoPLC
//     Main1_1 Outputs/Main1.Sequence1.Delta.internalKinChanPLCtoNC <-> Inputs/Main1.Sequence.Delta.internalKinChanPLCtoNC
//   ProjectMain/ProjectMain Instance <-> NC-Task 1 SAF/Objects/Delta MC CM
//     Main1_1 Inputs/Main1.Sequence1.Delta.internalCMGroup.NcToPlc <-> Group Outputs/ToPLC
//     Main1_1 Outputs/Main1.Sequence1.Delta.internalCMGroup.PlcToNc <-> Group Inputs/FromPLC
//   ProjectMain/ProjectMain Instance <-> NC-Task 1 SAF/Objects/Gantry MC CM
//     Main5_1 Inputs/GVL_XY.stGroupRef.NcToPlc <-> Group Outputs/ToPLC
//     Main5_1 Outputs/GVL_XY.stGroupRef.PlcToNc <-> Group Inputs/FromPLC

CONFIGURATION ProjectMain
    RESOURCE PLC ON TwinCAT3
        TASK Main1_1(INTERVAL := T#1ms, PRIORITY := 2);
        TASK Main2_1(INTERVAL := T#10ms, PRIORITY := 3);
        TASK Main3_1(INTERVAL := T#10ms, PRIORITY := 5);
        TASK Main4_1(INTERVAL := T#10ms, PRIORITY := 6);
        TASK Main5_1(INTERVAL := T#10ms, PRIORITY := 7);
        PROGRAM Main1 WITH Main1_1 : Main1;
        PROGRAM Main2 WITH Main2_1 : Main2;
        PROGRAM Main3 WITH Main3_1 : Main3;
        PROGRAM Main4 WITH Main4_1 : Main4;
        PROGRAM Main5 WITH Main5_1 : Main5;
    END_RESOURCE
END_CONFIGURATION

// ---- DUTs/DeltaCommands_typ.TcDUT
TYPE DeltaCommands_typ :
STRUCT
	
	ReturnHome			: BOOL;		// sends the delta to 0,0,0;
	PickFromElevator	: BOOL;		// Traverse to elevator, pick
	PlaceOnXTS			: BOOL;
	PickFromXTS			: BOOL;
	PlaceOnDump			: BOOL;
	EnableAutomatic		: BOOL;		// Starts the automatic process
	DisableAutomatic	: BOOL;		// Stops the automatic process
	
	TrackOnce			: BOOL;		// Track the next mover to pass the trigger then go home
	TrackContinuous		: BOOL;
	
	MoveDirectTo		: BOOL;		// 

END_STRUCT
END_TYPE

// ---- DUTs/DeltaMotionParameters_typ.TcDUT
TYPE DeltaMotionParameters_typ :
STRUCT
	
	Jerk			: LREAL;					// mm/s3
	Acceleration	: LREAL;					// mm/s2
	Deceleration	: LREAL;					// mm/s2
	Velocity		: LREAL;					// mm/s
	BlendingRadius	: LREAL;					// mm

END_STRUCT
END_TYPE

// ---- DUTs/DeltaState_enum.TcDUT
{attribute 'strict'}
TYPE DeltaState_enum :
(
	DL_IDLE				:= 0,	// Delta is idle, ungrouped, disabled
	DL_RESET			:= 10,	// Axes are reset to clear errors
	DL_POWER_AXES		:= 20,	// Axes are powered
	DL_SET_IK			:= 30,	// Inverse kinematics enabled
	DL_ADD_AXES_TO_CM	:= 40,	// Coordinated Motion group assembled
	DL_ENABLE_CM		:= 50,	// Enable CM Group
	DL_RUN				:= 60,	// Run Mode, ready for commands
	DL_DEBUG			:= 3113,
		
	DL_ERROR			:= 999
);
END_TYPE

// ---- DUTs/ElevatorState_enum.TcDUT
{attribute 'strict'}
TYPE ElevatorState_enum :
(	
	PE_IDLE			:= 0,
	PE_RESET		:= 10,
	PE_POWER_AXIS	:= 20,
	PE_RUN			:= 30,
	PE_DEBUG		:= 3113,
	PE_ERROR		:= 999
);
END_TYPE

// ---- DUTs/MachineOperationMode.TcDUT
TYPE MachineOperationMode :
STRUCT
	AUTO	: BOOL;
	MANUAL	: BOOL;
END_STRUCT
END_TYPE

// ---- DUTs/MainCommands_typ.TcDUT
TYPE MainCommands_typ :
STRUCT
	
	Enable		: BOOL;		// Enables Movers & Collision Avoidance, activates M1 Detection
	Start		: BOOL;		// Issues initial command, starts motion
	Stop		: BOOL;		// Stops movers, deregisters movers from all objectives	
	Disable		: BOOL;		// Disables Movers, Ungroups Movers
	
END_STRUCT
END_TYPE

// ---- DUTs/MainStateAxis_enum.TcDUT
{attribute 'strict'}
TYPE MainStateAxis_enum :
(
	MSA_DISABLED					:= 0,
	MSA_INITIALIZING				:= 10,
	MSA_ENABLING					:= 20,
	MSA_INITIALIZING_OBJECTIVES		:= 30,
	MSA_ENABLED						:= 40,
	MSA_RUN							:= 50,
	MSA_STOPPING					:= 60,
	MSA_STOPPED						:= 70,
	MSA_DISABLING					:= 80,
	MSA_ERROR						:= 90,
	MSA_DEBUG						:= 1000
);
END_TYPE

// ---- DUTs/MainState_enum.TcDUT
{attribute 'strict'}
TYPE MainState_enum :
(
	MS_DISABLED					:= 0,
	MS_INITIALIZING_MOVERS		:= 10,
	MS_ENABLING_MOVERS			:= 20,
	MS_INITIALIZING_OBJECTIVES	:= 30,
	MS_ENABLED					:= 40,
	MS_RUN						:= 50,
	MS_STOPPING					:= 60,
	MS_DISABLING				:= 70,
	MS_ERROR					:= 80,
	MS_STOPPED					:= 90,
	MS_DEBUG					:= 1000
);
END_TYPE

// ---- DUTs/MotionParameters_typ.TcDUT
TYPE MotionParameters_typ :
STRUCT
	
	Jerk			: LREAL;					// mm/s3
	Acceleration	: LREAL;					// mm/s2
	Deceleration	: LREAL;					// mm/s2
	Velocity		: LREAL;					// mm/s
	Direction		: Tc3_Mc3Definitions.MC_Direction;		// MC_Direction
	
END_STRUCT
END_TYPE

// ---- DUTs/MoverCommandType_enum.TcDUT
{attribute 'strict'}
TYPE MoverCommandType_enum :
(
	MOVETYPE_NONE		:= 0,
	MOVETYPE_POSITION	:= 1,
	MOVETYPE_STATION	:= 2,
	MOVETYPE_VELOCITY	:= 3,
	MOVETYPE_SYNC		:= 4
);
END_TYPE

// ---- DUTs/MoverState_enum.TcDUT
{attribute 'strict'}
TYPE MoverState_enum :
(
	MV_IDLE				:= 0,
	MV_RESET			:= 10,
	MV_M1_READMODE		:= 20,
	MV_M1_EVALMODE		:= 30,
	MV_M1_READSTATUS	:= 40,
	MV_M1_EVALSTATUS	:= 50,
	MV_M1_DETECT		:= 60,
	MV_ENABLING			:= 70,
	MV_ADDTOGROUP		:= 80,
	MV_READGROUPSTATUS	:= 90,
	MV_RESETGROUP		:= 100,
	MV_ENABLEGROUP		:= 110,
	MV_RUN				:= 120,
	MV_REMOVEFROMGROUP	:= 130,
	MV_BEGIN_HALTING	:= 140,
	MV_HALTING			:= 150,
	MV_DISABLING		:= 160,
	MV_ERROR			:= 999
);
END_TYPE

// ---- DUTs/MoveState_t.TcDUT
TYPE MoveState_t :
(
	MOVESTATE_INIT,
	MOVESTATE_ENABLE,
	MOVESTATE_FORWARD,
	MOVESTATE_BACKWARDS,
	MOVESTATE_BACKWARDSSLOW,
	MOVESTATE_NEWTARGETPOSITION,
	MOVESTATE_ERROR,
	MOVESTATE_STOP,
	MOVESTATE_RESET
	
)UDINT;
END_TYPE

// ---- DUTs/PickPars_typ.TcDUT
TYPE PickPars_typ :
STRUCT
	
	PlaceXTS	: Vector3Position_typ;
	Elevator	: Vector3Position_typ;
	Conveyer 	: Vector3Position_typ;
	HomePos		: Vector3Position_typ;
	DumpPos		: Vector3Position_typ;
	LoadTime	: TIME;
	UnloadTime	: TIME;

END_STRUCT
END_TYPE

// ---- DUTs/Pucks.TcDUT
TYPE Pucks :
STRUCT
	y 		 	: LREAL;
	zOffset		: LREAL;
	xOffset		: LREAL;
	code	 	: INT;
END_STRUCT
END_TYPE

// ---- DUTs/SystemCommands_typ.TcDUT
TYPE SystemCommands_typ :
STRUCT
	
	MoverRelease		: BOOL;	// release a mover from the delta place position
	
	EnableTimerRelease	: BOOL;	// automatically releases movers from delta on a timer

	Delta				: DeltaCommands_typ;
	
	ReloadElevator		: BOOL;	// sets the elevator to a zero position and refreshes the puck count

END_STRUCT
END_TYPE

// ---- DUTs/Vector3Position_typ.TcDUT
TYPE Vector3Position_typ :
STRUCT
	X		: LREAL;
	Y		: LREAL;
	Z		: LREAL;
END_STRUCT
END_TYPE

// ---- DUTs/Visu_typ.TcDUT
TYPE Visu_typ :
STRUCT
	
	MoveDirect_X		: LREAL;
	MoveDirect_Y		: LREAL;
	MoveDirect_Z 		: LREAL;

END_STRUCT
END_TYPE

// ---- DUTs/Coords.TcDUT
TYPE Coords :
STRUCT
	sName : STRING;
	iID 	: INT;
	x	: LREAL;
	y	: LREAL;
	z	: LREAL;
END_STRUCT
END_TYPE

// ---- DUTs/XYParams_typ.TcDUT
TYPE XYParams_typ :
STRUCT
	bUserIncrementStep		: BOOL;
	bUserInfiniteMovement 	: BOOL; 
	nState					: INT;
	nNextState				: INT;
	fVelFactor				: LREAL;
END_STRUCT
END_TYPE

// ---- GVLs/GVL.TcGVL
{attribute 'qualified_only'}
VAR_GLOBAL
	bGantryVac 			AT %Q*:BOOL;
	bGantryDown 		AT %Q*:BOOL;
	bGantryUp 			AT %Q*:BOOL;
	bLoadNewPuck		: BOOL;
	Pucks				: ARRAY[0..39] OF Pucks;
	puckIncrement		: INT := 0;
	bClearPuck			: BOOL;
	bPuckMissed			: BOOL;
	iMissedPucks		: INT := 0;
	iPucksPicked		: INT := 0;
	bDumpPuck			: BOOL;
END_VAR

VAR_GLOBAL PERSISTENT
 	DeltaCoords 		: ARRAY[0..20] OF Coords;
	XYCoords			: ARRAY[0..20] OF Coords;
	iMovementNumber		:INT;
END_VAR

// ---- GVLs/GVL_Conveyer.TcGVL
{attribute 'qualified_only'}
VAR_GLOBAL
	ConveyerAxis 			: AXIS_REF;
	bConveyerReadyToMove 	: BOOL;
	bConveyerReadyToPick 	: BOOL;
	bSensor 				AT %I*: BOOL;
END_VAR

// ---- GVLs/GVL_Vision.TcGVL
{attribute 'qualified_only'}
VAR_GLOBAL

	cmdTrigCamera	: BOOL;
	outputValid		: BOOL;
	noRead			: BOOL;
	PuckValue		: INT;

END_VAR

// ---- GVLs/GVL_XTS.TcGVL
{attribute 'qualified_only'}
VAR_GLOBAL
	bDeltaRelease 		AT %Q* : BOOL;
	bDeltaReleased 		AT %I* : BOOL;
	mover0InPosition 	AT %I* : BOOL;
	moversInPosition	AT %I* : ARRAY [1..3] OF BOOL;
	moversReleased		AT %I* : ARRAY [1..3] OF BOOL;
	moversRelease		AT %Q* : ARRAY [1..3] OF BOOL;
	
	XTS_Enable				AT %Q* : BOOL;
	XTS_Start				AT %Q* : BOOL;
	XTS_Stop				AT %Q* : BOOL;
	XTS_Disable				AT %Q* : BOOL;
	
END_VAR

// ---- GVLs/GVL_XY.TcGVL
{attribute 'qualified_only'}
VAR_GLOBAL
    stGroupRef            	: AXES_GROUP_REF;
    stAxis                	: ARRAY[1..cAxesCount] OF AXIS_REF;
	stSlaveAxis				: ARRAY[1..cAxesSlaveCount] of AXIS_REF;
	bAirEnable				AT %Q* : BOOL;
	bPushDown				AT %Q* : BOOL;
	bPullUp					AT %Q* : BOOL;
END_VAR

VAR_GLOBAL CONSTANT
    cAxesCount            	: UINT:=2;
	cAxesSlaveCount			: UINT:=1;
END_VAR

// ---- ITFs/iDelta.TcIO
INTERFACE iDelta

METHOD ExecuteRoute : BOOL
VAR_INPUT
END_VAR
END_METHOD

METHOD MoveDirectTo : BOOL
VAR_INPUT
END_VAR
END_METHOD

METHOD MoveX : BOOL
VAR_INPUT
END_VAR
END_METHOD

METHOD MoveY : BOOL
VAR_INPUT
END_VAR
END_METHOD

METHOD MoveZ : BOOL
VAR_INPUT
END_VAR
END_METHOD

METHOD ReturnHome : BOOL
VAR_INPUT
END_VAR
END_METHOD

METHOD SetAcceleration : BOOL
VAR_INPUT
	Acceleration	: LREAL;
END_VAR
END_METHOD

METHOD SetDeceleration : BOOL
VAR_INPUT
END_VAR
END_METHOD

METHOD SetJerk : BOOL
VAR_INPUT
END_VAR
END_METHOD

METHOD SetVelocity : BOOL
VAR_INPUT
END_VAR
END_METHOD

METHOD TraverseAtHeightTo : BOOL
VAR_INPUT
END_VAR
END_METHOD

END_INTERFACE

// ---- ITFs/iRoute.TcIO
INTERFACE iRoute

METHOD AddBlendedPoint : iRoute
VAR_INPUT
	X			: LREAL;
	Y			: LREAL;
	Z			: LREAL;
END_VAR
END_METHOD

METHOD AddViaPoint : iRoute
VAR_INPUT
	X			: LREAL;
	Y			: LREAL;
	Z			: LREAL;
END_VAR
END_METHOD

METHOD ClearRoute : iRoute
VAR_INPUT
END_VAR
END_METHOD

END_INTERFACE
